// Copyright (c) 2024 Loupe (https://loupe.team), provided under the MIT License.
TYPE STRING_EX_LEN : STRING(2000); END_TYPE

(* stored: Version 1.1.0.1, ProductVersion 3.1.4024.12
   DUT STRING_EX_LEN: Id {ee5ab662-46b9-48e0-aa78-fcaad380107f} *)
